% RSLogix 500 project ROTATOMETER.RSS, saved by version 8.30.00.16 %
PROJECT "UNTITLED"    % processor: Bul.1763 MicroLogix 1100 Series B %

PROGRAM FILES
  LAD 2 "MAIN"  3 rungs
  LAD 3 "CONTROL"  6 rungs

DATA FILES
  O0 OUTPUT  5 elements
  I1 INPUT  7 elements
  S2 STATUS  66 elements
  B3 BINARY  1 elements
  T4 TIMER  1 elements
  C5 COUNTER  1 elements
  R6 CONTROL  1 elements
  N7 INTEGER  3 elements
  F8 FLOAT  2 elements

LADDER 2 "MAIN"
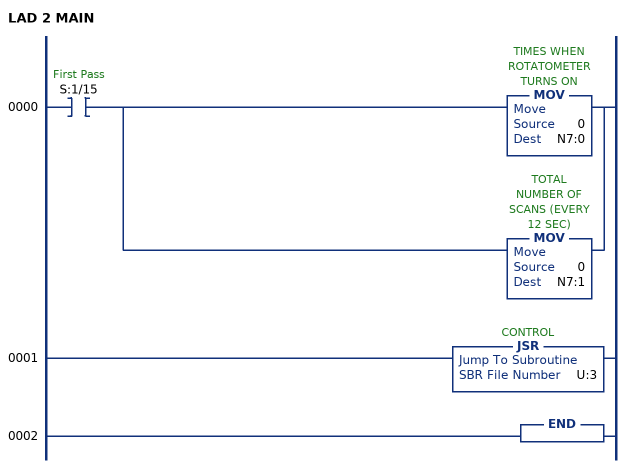
% Rung: 0 %
SOR XIC S:1/15 BST MOV 0 N7:0 NXB MOV 0 N7:1 BND EOR
%   S:1/15  "First Pass" %
%   N7:0  "TIMES WHEN ROTATOMETER TURNS ON" %
%   N7:1  "TOTAL NUMBER OF SCANS (EVERY 12 SEC)" %
% Rung: 1 %
SOR JSR U:3 EOR
%   U:3  "CONTROL" %
% Rung: 2 %
SOR END EOR

LADDER 3 "CONTROL"
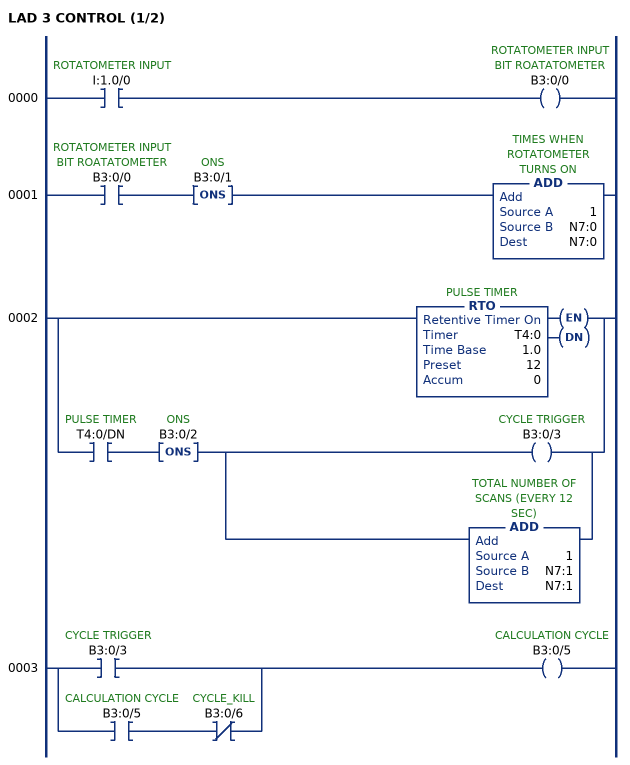
% Rung: 0 %
SOR XIC I:1.0/0 OTE B3:0/0 EOR
%   I:1.0/0  "ROTATOMETER INPUT" %
%   B3:0/0  ROATATOMETER  "ROTATOMETER INPUT BIT" %
% Rung: 1 %
SOR XIC B3:0/0 ONS B3:0/1 ADD 1 N7:0 N7:0 EOR
%   B3:0/0  ROATATOMETER  "ROTATOMETER INPUT BIT" %
%   B3:0/1  "ONS" %
%   N7:0  "TIMES WHEN ROTATOMETER TURNS ON" %
% Rung: 2 %
SOR BST RTO T4:0 1.0 12 0 NXB XIC T4:0/DN ONS B3:0/2 BST OTE B3:0/3 NXB ADD 1 N7:1 N7:1 BND BND EOR
%   T4:0  "PULSE TIMER" %
%   T4:0/DN  "PULSE TIMER" %
%   B3:0/2  "ONS" %
%   B3:0/3  "CYCLE TRIGGER" %
%   N7:1  "TOTAL NUMBER OF SCANS (EVERY 12 SEC)" %
% Rung: 3 %
SOR BST XIC B3:0/3 NXB XIC B3:0/5 XIO B3:0/6 BND OTE B3:0/5 EOR
%   B3:0/3  "CYCLE TRIGGER" %
%   B3:0/5  "CALCULATION CYCLE" %
%   B3:0/6  "CYCLE_KILL" %

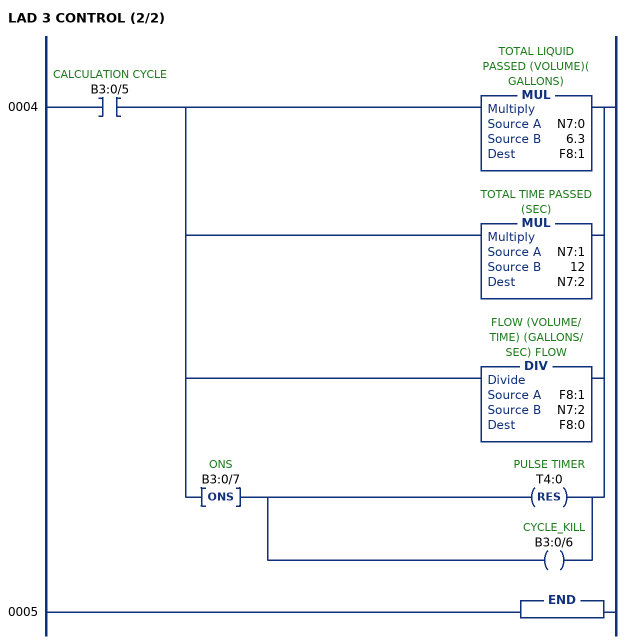
% Rung: 4 %
SOR XIC B3:0/5 BST MUL N7:0 6.3 F8:1 NXB MUL N7:1 12 N7:2 NXB DIV F8:1 N7:2 F8:0 NXB ONS B3:0/7 BST RES T4:0 NXB OTE B3:0/6 BND BND EOR
%   B3:0/5  "CALCULATION CYCLE" %
%   N7:0  "TIMES WHEN ROTATOMETER TURNS ON" %
%   F8:1  "TOTAL LIQUID PASSED (VOLUME)(GALLONS)" %
%   N7:1  "TOTAL NUMBER OF SCANS (EVERY 12 SEC)" %
%   N7:2  "TOTAL TIME PASSED (SEC)" %
%   F8:0  FLOW  "FLOW (VOLUME/TIME) (GALLONS/SEC)" %
%   B3:0/7  "ONS" %
%   T4:0  "PULSE TIMER" %
%   B3:0/6  "CYCLE_KILL" %
% Rung: 5 %
SOR END EOR

OTHER DOCUMENTED ADDRESSES
  B3:0/4  "TIMER RESET"
  I:0.0/0  "ROTATOMETER INPUT"

DATA TABLE (non-zero values as saved)
DATA T4
% .PRE .ACC %
% T4:0 % 12 0
